// TIA Portal V16 export
// export: Created 2021-06-28T08:13:57.7608914Z, ExportSetting WithDefaults, DisplayName Totally Integrated Automation Portal, DisplayVersion V16 Update 4, DisplayName TIA Portal Version Control Interface, DisplayVersion V16 Update 2, DisplayName TIA Portal Openness, DisplayVersion V16 Update 4, DisplayName STEP 7 Professional, DisplayVersion V16 Update 4, DisplayName STEP 7 Safety, DisplayVersion V16, DisplayName WinCC Advanced, DisplayVersion V16 Update 4
FUNCTION "Actuator_Interlock" : Void   // FC3, LAD
{ S7_Optimized_Access := 'TRUE' }
VERSION : 0.1
// stored: AutoNumber true, IsIECCheckEnabled false, SetENOAutomatically false, UDAEnableTagReadback false
   VAR_TEMP   // added for the SCL form of the ladder/FBD networks
      _w1 : Bool;
   END_VAR
BEGIN

REGION Network 1
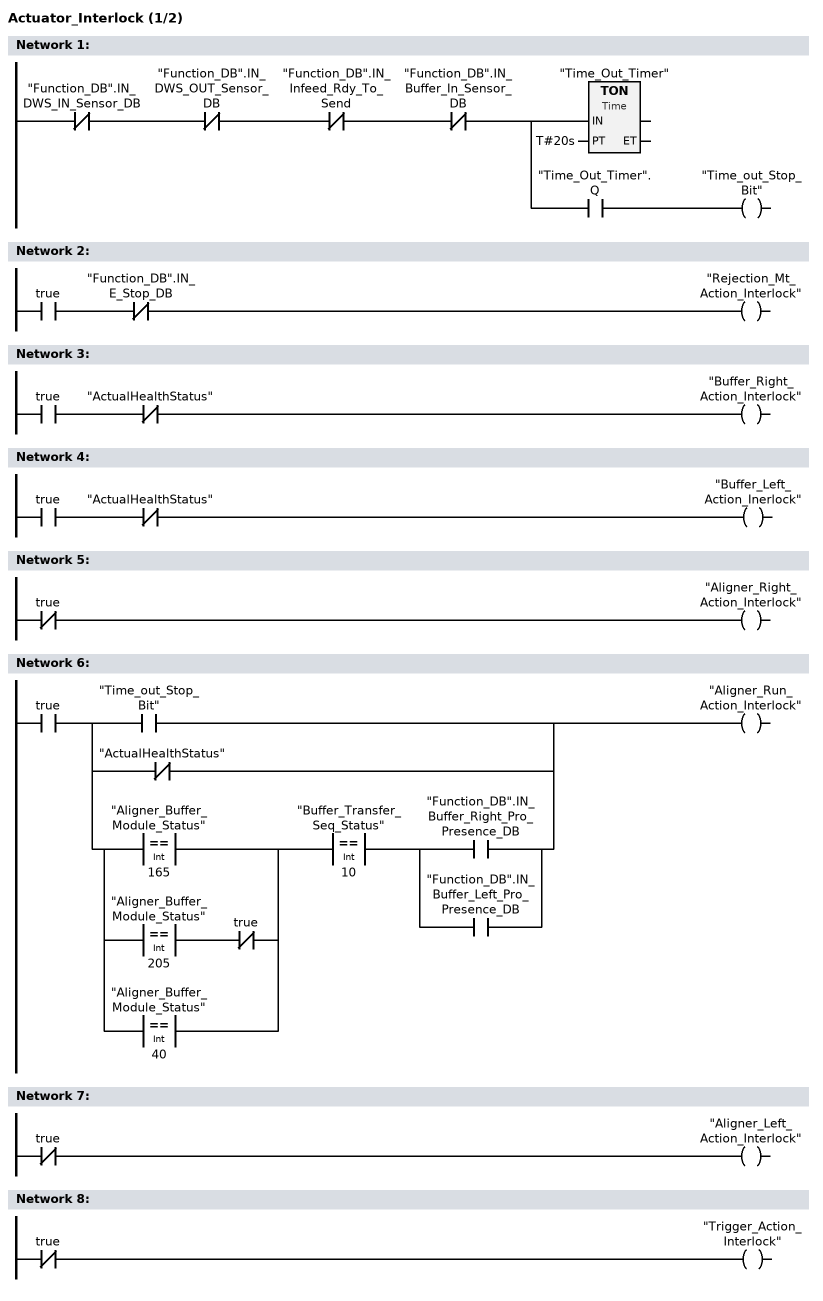
   RUNG wire#powerrail
      I_Contact( "Function_DB".IN_DWS_IN_Sensor_DB )
      I_Contact( "Function_DB".IN_DWS_OUT_Sensor_DB )
      I_Contact( "Function_DB".IN_Infeed_Rdy_To_Send )
      I_Contact( "Function_DB".IN_Buffer_In_Sensor_DB )
      wire#w1
      { S7_Templates := "time_type := Time" } "Time_Out_Timer".TON(pt := T#20s, et =>)
   END_RUNG
   RUNG wire#w1
      Contact( "Time_Out_Timer".Q )
      Coil( "Time_out_Stop_Bit" )
   END_RUNG
   // the same network as SCL:
   #_w1 := NOT "Function_DB".IN_DWS_IN_Sensor_DB AND NOT "Function_DB".IN_DWS_OUT_Sensor_DB AND NOT "Function_DB".IN_Infeed_Rdy_To_Send AND NOT "Function_DB".IN_Buffer_In_Sensor_DB;
   "Time_Out_Timer".TON(IN := #_w1, PT := T#20s);
   "Time_out_Stop_Bit" := #_w1 AND "Time_Out_Timer".Q;
END_REGION

REGION Network 2
   RUNG wire#powerrail
      Contact( true )
      I_Contact( "Function_DB".IN_E_Stop_DB )
      Coil( "Rejection_Mt_Action_Interlock" )
   END_RUNG
   // the same network as SCL:
   "Rejection_Mt_Action_Interlock" := true AND NOT "Function_DB".IN_E_Stop_DB;
END_REGION

REGION Network 3
   RUNG wire#powerrail
      Contact( true )
      I_Contact( "ActualHealthStatus" )
      Coil( "Buffer_Right_Action_Interlock" )
   END_RUNG
   // the same network as SCL:
   "Buffer_Right_Action_Interlock" := true AND NOT "ActualHealthStatus";
END_REGION

REGION Network 4
   RUNG wire#powerrail
      Contact( true )
      I_Contact( "ActualHealthStatus" )
      Coil( "Buffer_Left_Action_Inerlock" )
   END_RUNG
   // the same network as SCL:
   "Buffer_Left_Action_Inerlock" := true AND NOT "ActualHealthStatus";
END_REGION

REGION Network 5
   RUNG wire#powerrail
      I_Contact( true )
      Coil( "Aligner_Right_Action_Interlock" )
   END_RUNG
   // the same network as SCL:
   "Aligner_Right_Action_Interlock" := NOT true;
END_REGION

REGION Network 6
   RUNG wire#powerrail
      Contact( true )
      wire#w1
      Contact( "Time_out_Stop_Bit" )
      wire#w2
      Coil( "Aligner_Run_Action_Interlock" )
   END_RUNG
   RUNG wire#w1
      I_Contact( "ActualHealthStatus" )
   END_RUNG wire#w2
   RUNG wire#w1
      { S7_Templates := "SrcType := Int" } EQ_Contact(in1 := "Aligner_Buffer_Module_Status", in2 := 165)
      wire#w3
      { S7_Templates := "SrcType := Int" } EQ_Contact(in1 := "Buffer_Transfer_Seq_Status", in2 := 10)
      wire#w4
      Contact( "Function_DB".IN_Buffer_Right_Pro_Presence_DB )
   END_RUNG wire#w2
   RUNG wire#w1
      { S7_Templates := "SrcType := Int" } EQ_Contact(in1 := "Aligner_Buffer_Module_Status", in2 := 205)
      I_Contact( true )
   END_RUNG wire#w3
   RUNG wire#w1
      { S7_Templates := "SrcType := Int" } EQ_Contact(in1 := "Aligner_Buffer_Module_Status", in2 := 40)
   END_RUNG wire#w3
   RUNG wire#w4
      Contact( "Function_DB".IN_Buffer_Left_Pro_Presence_DB )
   END_RUNG wire#w2
   // the same network as SCL:
   "Aligner_Run_Action_Interlock" := true AND ("Time_out_Stop_Bit" OR NOT "ActualHealthStatus" OR ((("Aligner_Buffer_Module_Status" = 165) OR (("Aligner_Buffer_Module_Status" = 205) AND NOT true) OR ("Aligner_Buffer_Module_Status" = 40)) AND ("Buffer_Transfer_Seq_Status" = 10) AND ("Function_DB".IN_Buffer_Right_Pro_Presence_DB OR "Function_DB".IN_Buffer_Left_Pro_Presence_DB)));
END_REGION

REGION Network 7
   RUNG wire#powerrail
      I_Contact( true )
      Coil( "Aligner_Left_Action_Interlock" )
   END_RUNG
   // the same network as SCL:
   "Aligner_Left_Action_Interlock" := NOT true;
END_REGION

REGION Network 8
   RUNG wire#powerrail
      I_Contact( true )
      Coil( "Trigger_Action_Interlock" )
   END_RUNG
   // the same network as SCL:
   "Trigger_Action_Interlock" := NOT true;
END_REGION

REGION Network 9
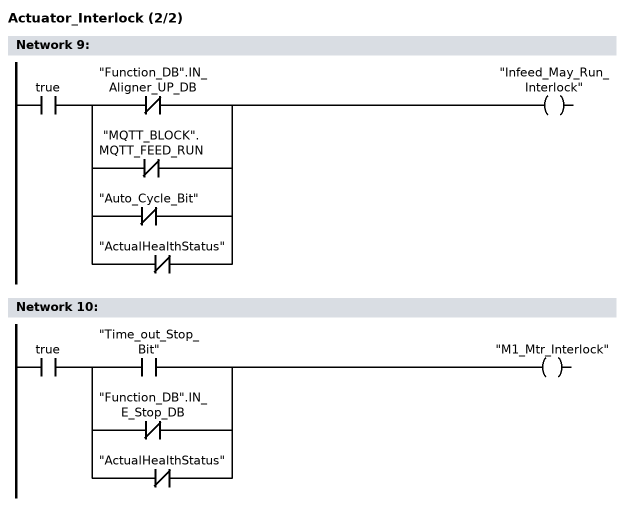
   RUNG wire#powerrail
      Contact( true )
      wire#w1
      I_Contact( "Function_DB".IN_Aligner_UP_DB )
      wire#w2
      Coil( "Infeed_May_Run_Interlock" )
   END_RUNG
   RUNG wire#w1
      I_Contact( "MQTT_BLOCK".MQTT_FEED_RUN )
   END_RUNG wire#w2
   RUNG wire#w1
      I_Contact( "Auto_Cycle_Bit" )
   END_RUNG wire#w2
   RUNG wire#w1
      I_Contact( "ActualHealthStatus" )
   END_RUNG wire#w2
   // the same network as SCL:
   "Infeed_May_Run_Interlock" := true AND (NOT "Function_DB".IN_Aligner_UP_DB OR NOT "MQTT_BLOCK".MQTT_FEED_RUN OR NOT "Auto_Cycle_Bit" OR NOT "ActualHealthStatus");
END_REGION

REGION Network 10
   RUNG wire#powerrail
      Contact( true )
      wire#w1
      Contact( "Time_out_Stop_Bit" )
      wire#w2
      Coil( "M1_Mtr_Interlock" )
   END_RUNG
   RUNG wire#w1
      I_Contact( "Function_DB".IN_E_Stop_DB )
   END_RUNG wire#w2
   RUNG wire#w1
      I_Contact( "ActualHealthStatus" )
   END_RUNG wire#w2
   // the same network as SCL:
   "M1_Mtr_Interlock" := true AND ("Time_out_Stop_Bit" OR NOT "Function_DB".IN_E_Stop_DB OR NOT "ActualHealthStatus");
END_REGION
END_FUNCTION
